TYPE SmokeControlExerciseParameters :
STRUCT
	Interval: INT := 48; (* Central exercise interval for all damper modules (set to zero for no exercising) $(unit hour) *)
	StopVentilation: BOOL := TRUE; (* Stop ventilation during central exercise *)
	Hour: INT := 10; (* Central exercise at this hour $(unit hour) *)
	Minute: INT := 30; (* Central exercise at this minute $(unit minute) *)
END_STRUCT
END_TYPE

(* stored: Version 1.1.0.1, ProductVersion 3.1.4024.6
   DUT SmokeControlExerciseParameters: Id {e404acbd-2aa5-4c64-b4cc-59e95421f5aa} *)
